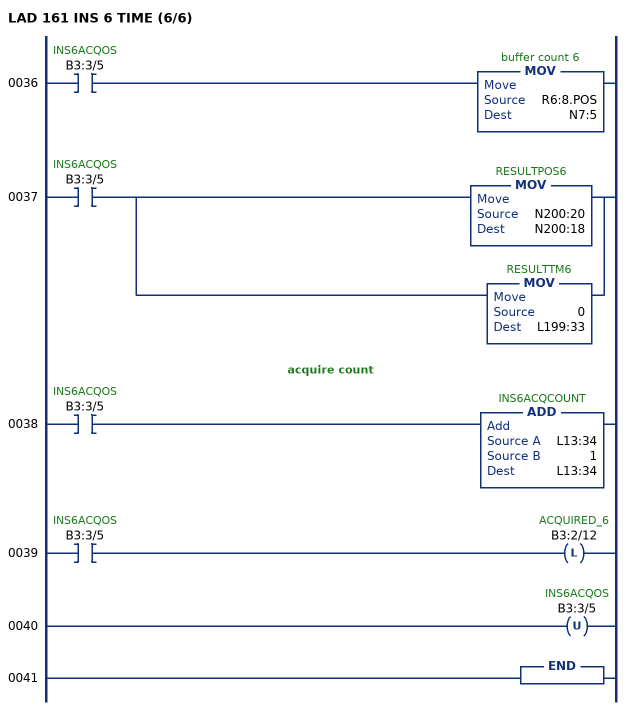
% Rung: 36 %
SOR XIC B3:3/5 MOV R6:8.POS N7:5 EOR
%   B3:3/5  INS6ACQOS %
%   R6:8  "track part location until acquire 6" %
%   N7:5  "buffer count 6" %
% Rung: 37 %
SOR XIC B3:3/5 BST MOV N200:20 N200:18 NXB MOV 0 L199:33 BND EOR
%   B3:3/5  INS6ACQOS %
%   N200:20  ACQPOS6  "part acq pos 6" %
%   N200:18  RESULTPOS6 %
%   L199:33  RESULTTM6 %
% Rung: 38 %
% TITLE: acquire count %
SOR XIC B3:3/5 ADD L13:34 1 L13:34 EOR
%   B3:3/5  INS6ACQOS %
%   L13:34  INS6ACQCOUNT %
% Rung: 39 %
SOR XIC B3:3/5 OTL B3:2/12 EOR
%   B3:3/5  INS6ACQOS %
%   B3:2/12  ACQUIRED_6 %
% Rung: 40 %
SOR OTU B3:3/5 EOR
%   B3:3/5  INS6ACQOS %
% Rung: 41 %
SOR END EOR

LADDER 162 "INS 6 NEW"
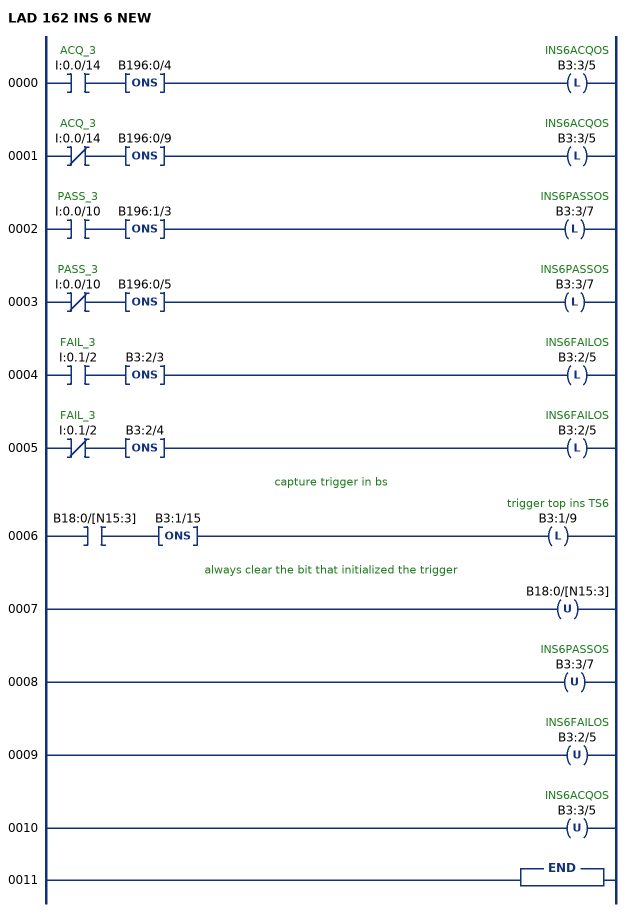
% Rung: 0 %
SOR XIC I:0.0/14 ONS B196:0/4 OTL B3:3/5 EOR
%   I:0.0/14  ACQ_3 %
%   B3:3/5  INS6ACQOS %
% Rung: 1 %
SOR XIO I:0.0/14 ONS B196:0/9 OTL B3:3/5 EOR
%   I:0.0/14  ACQ_3 %
%   B3:3/5  INS6ACQOS %
% Rung: 2 %
SOR XIC I:0.0/10 ONS B196:1/3 OTL B3:3/7 EOR
%   I:0.0/10  PASS_3 %
%   B3:3/7  INS6PASSOS %
% Rung: 3 %
SOR XIO I:0.0/10 ONS B196:0/5 OTL B3:3/7 EOR
%   I:0.0/10  PASS_3 %
%   B3:3/7  INS6PASSOS %
% Rung: 4 %
SOR XIC I:0.1/2 ONS B3:2/3 OTL B3:2/5 EOR
%   I:0.1/2  FAIL_3 %
%   B3:2/5  INS6FAILOS %
% Rung: 5 %
SOR XIO I:0.1/2 ONS B3:2/4 OTL B3:2/5 EOR
%   I:0.1/2  FAIL_3 %
%   B3:2/5  INS6FAILOS %
% Rung: 6 %
% capture trigger in bs %
SOR XIC B18:0/[N15:3] ONS B3:1/15 OTL B3:1/9 EOR
%   N15:3  INS_6_TRIG_LOC %
%   B3:1/9  TS6  "trigger top ins" %
% Rung: 7 %
% always clear the bit that initialized the trigger %
SOR OTU B18:0/[N15:3] EOR
%   N15:3  INS_6_TRIG_LOC %
% Rung: 8 %
SOR OTU B3:3/7 EOR
%   B3:3/7  INS6PASSOS %
% Rung: 9 %
SOR OTU B3:2/5 EOR
%   B3:2/5  INS6FAILOS %
% Rung: 10 %
SOR OTU B3:3/5 EOR
%   B3:3/5  INS6ACQOS %
% Rung: 11 %
SOR END EOR

LADDER 170 "PASS BLOW"
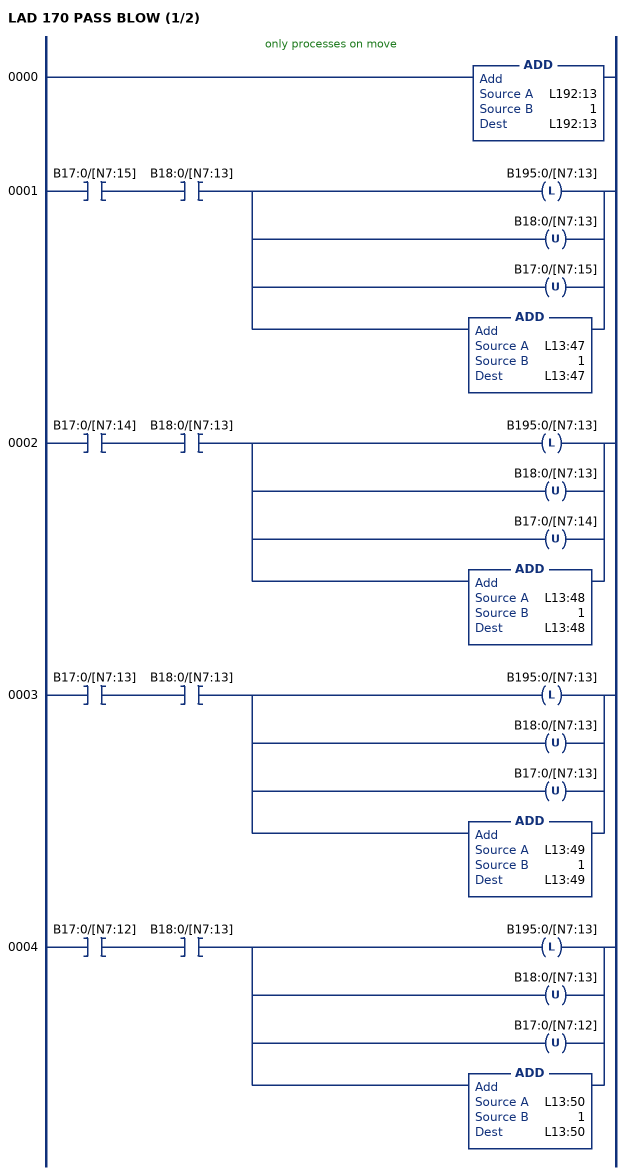
% Rung: 0 %
% only processes on move %
SOR ADD L192:13 1 L192:13 EOR
% Rung: 1 %
SOR XIC B17:0/[N7:15] XIC B18:0/[N7:13] BST OTL B195:0/[N7:13] NXB OTU B18:0/[N7:13] NXB OTU B17:0/[N7:15] NXB ADD L13:47 1 L13:47 BND EOR
%   N7:15  OS5 %
%   N7:13  OS3 %
% Rung: 2 %
SOR XIC B17:0/[N7:14] XIC B18:0/[N7:13] BST OTL B195:0/[N7:13] NXB OTU B18:0/[N7:13] NXB OTU B17:0/[N7:14] NXB ADD L13:48 1 L13:48 BND EOR
%   N7:14  OS4 %
%   N7:13  OS3 %
% Rung: 3 %
SOR XIC B17:0/[N7:13] XIC B18:0/[N7:13] BST OTL B195:0/[N7:13] NXB OTU B18:0/[N7:13] NXB OTU B17:0/[N7:13] NXB ADD L13:49 1 L13:49 BND EOR
%   N7:13  OS3 %
% Rung: 4 %
SOR XIC B17:0/[N7:12] XIC B18:0/[N7:13] BST OTL B195:0/[N7:13] NXB OTU B18:0/[N7:13] NXB OTU B17:0/[N7:12] NXB ADD L13:50 1 L13:50 BND EOR
%   N7:12  OS2 %
%   N7:13  OS3 %

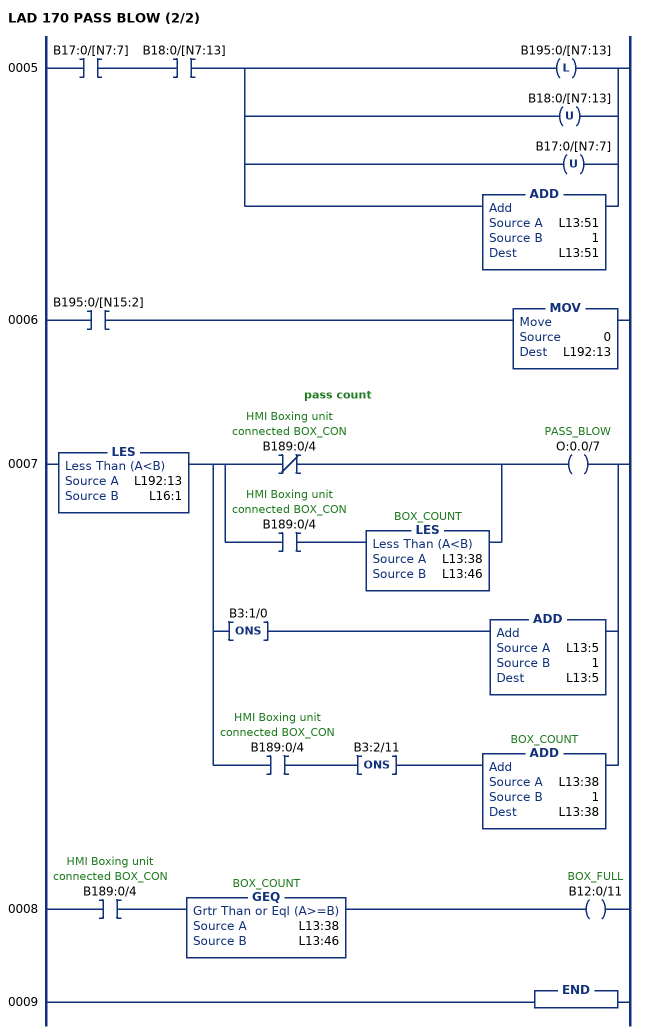
% Rung: 5 %
SOR XIC B17:0/[N7:7] XIC B18:0/[N7:13] BST OTL B195:0/[N7:13] NXB OTU B18:0/[N7:13] NXB OTU B17:0/[N7:7] NXB ADD L13:51 1 L13:51 BND EOR
%   N7:7  OS1 %
%   N7:13  OS3 %
% Rung: 6 %
SOR XIC B195:0/[N15:2] MOV 0 L192:13 EOR
%   N15:2  BLOW_PT %
% Rung: 7 %
% TITLE: pass count %
SOR LES L192:13 L16:1 BST BST XIO B189:0/4 NXB XIC B189:0/4 LES L13:38 L13:46 BND OTE O:0.0/7 NXB ONS B3:1/0 ADD L13:5 1 L13:5 NXB XIC B189:0/4 ONS B3:2/11 ADD L13:38 1 L13:38 BND EOR
%   L16:1  BLOW_TIME %
%   B189:0/4  BOX_CON  "HMI Boxing unit connected" %
%   L13:38  BOX_COUNT %
%   L13:46  BOX_LIMIT  "box count setpoint" %
%   O:0.0/7  PASS_BLOW %
% Rung: 8 %
SOR XIC B189:0/4 GEQ L13:38 L13:46 OTE B12:0/11 EOR
%   B189:0/4  BOX_CON  "HMI Boxing unit connected" %
%   L13:38  BOX_COUNT %
%   L13:46  BOX_LIMIT  "box count setpoint" %
%   B12:0/11  BOX_FULL %
% Rung: 9 %
SOR END EOR

LADDER 180 "RATE"
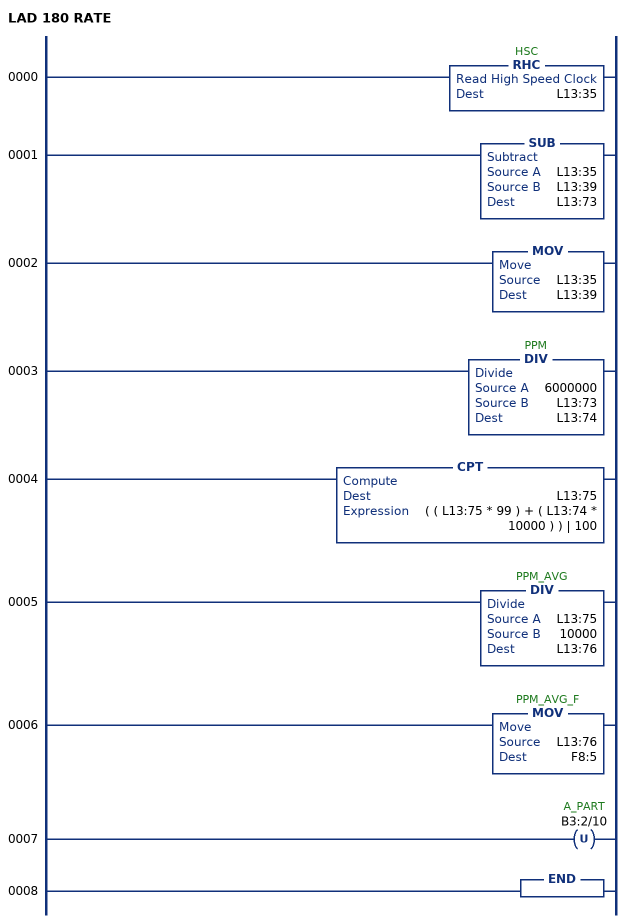
% Rung: 0 %
SOR RHC L13:35 EOR
%   L13:35  HSC %
% Rung: 1 %
SOR SUB L13:35 L13:39 L13:73 EOR
%   L13:35  HSC %
% Rung: 2 %
SOR MOV L13:35 L13:39 EOR
%   L13:35  HSC %
% Rung: 3 %
SOR DIV 6000000 L13:73 L13:74 EOR
%   L13:74  PPM %
% Rung: 4 %
SOR CPT L13:75 " ( ( L13:75 * 99 ) + ( L13:74 * 10000 ) ) | 100 " EOR
%   L13:74  PPM %
% Rung: 5 %
SOR DIV L13:75 10000 L13:76 EOR
%   L13:76  PPM_AVG %
% Rung: 6 %
SOR MOV L13:76 F8:5 EOR
%   L13:76  PPM_AVG %
%   F8:5  PPM_AVG_F %
% Rung: 7 %
SOR OTU B3:2/10 EOR
%   B3:2/10  A_PART %
% Rung: 8 %
SOR END EOR

OTHER DOCUMENTED ADDRESSES
  B3:4/12  "trig 1 event"
  B3:5/1  "placeholder"
  B3:8/1  "bypass extra trigger camera 2"
  B3:8/2  "bypass extra trigger camera 3"
  B3:8/3  "bypass extra trigger camera 4"
  B3:8/6  "a bypass bit"
  B3:8/7  "a bypass bit"
  B3:8/12  "start bottom top camera responce"
  B3:8/13  "extra blow signal for testing"
  B3:8/15  "start side camera responce"
  B3:9/2  "one shot"
  B3:9/4  "start top camera responce"
  B3:9/6  "C1D"
  B3:9/7  "C1t"
  B3:9/8  "C2D"
  B3:9/9  "C2t"
  B3:9/14  "input from hmi to reset count"
  B3:10/0  "bypass part too close"
  B3:10/2  "One Shot"
  B3:10/3  "One Shot"
  B3:10/4  "changing Box chute door operation"
  B3:10/5  "one shot"
  B3:10/6  "excessive data output time"
  B3:10/9  "one shot"
  B3:10/10  "one shot"
  B3:10/11  "bottom part present trailling edge"
  B3:10/13  "one shot"
  B3:10/14  "Dont use"
  B3:10/15  "Reserved For Shift Registers"
  B3:11/0  "bypass unused portion of code"
  B3:11/1  "bypass"
  B3:11/2  "Enable encoder belt movement simulation when testing"
  B3:11/3  "Block blow signals while changing box"
  B3:11/4  "one shot"
  B3:11/6  "one shot"
  B3:11/7  "one shot"
  B3:11/8  "one shot"
  B3:11/11  "one shot"
  B3:11/12  "one shot"
  B3:11/15  "one shot"
  B3:12/0  "one shot"
  B3:12/1  "one shot"
  B3:12/2  "Command 2 Oneshot"
  B3:12/3  "Command 2 Active"
  B3:12/4  "Command3 Oneshot"
  B3:12/5  "Command 3 Active"
  B3:12/6  "Inspection Command Counter"
  B3:12/7  "Command 4 Active"
  B3:12/8  "Command 4 Oneshot"
  B3:12/14  "flip flop bit"
  B3:13/5  "bypass"
  B3:13/6  "Off"
  B3:13/7  "On"
  B3:13/8  "On"
  B3:13/9  "Off"
  B3:13/10  "On"
  B3:13/11  "Off"
  B3:13/12  "Test Trigger to laser Spacing"
  B3:13/15  "Test Signals"
  B3:17/12  "Always Off"
  B9:0/0  "Trigger Insert Position"
  B9:0/1  "bottom of top conveyor part transfer location"
  B9:0/[N7:0]  "Side Camera Trigger Posistion"
  B9:0/[N7:2]  "Mask Start Position"
  B9:0/[N7:6]  "Blow Off Position"
  B9:0/[N7:20]  "part present bit shift load position"
  B9:0/[N7:48]  "Top Camera Trigger Posistion"
  B9:0/[N16:0]  "Trigger Position"
  B9:0/[N17:8]  "part from bottom belt present at top belt optic position"
  B10:0/0  "Pass Insert Position"
  B10:0/[N7:2]  "Pass Bit Position"
  B10:0/[N7:4]  "Pass Insert Position"
  B10:0/[N7:5]  "Pass Start Position"
  B10:0/[N7:6]  "Pass Position"
  B10:0/[N16:4]  "Pass Insert Position"
  B10:0/[N16:6]  "Pass Position"
  B11:0/0  "Trigger Insert Position"
  B11:0/[N7:8]  "Fail Bit Position"
  B11:0/[N16:0]  "Trigger Position"
  B12:1/0  "Conveyor Start Oneshot"
  B12:1/1  "Feed Start Oneshot"
  B12:1/2  "Conveyor Stop Oneshot"
  B12:1/3  "Feed Stop Oneshot"
  B12:1/5  "Conveyor Start Oneshot"
  B12:10  BULK_PACK
  B14:0/0  "Bottom Pass Insert"
  B14:0/4  "Bottom Pass Insert Position"
  B14:0/[N13:14]  "Start Laser Pass"
  B14:0/[N16:4]  "Pass Insert Position"
  B14:0/[N16:6]  "Pass Position"
  B15:0  "Alarm Bits"
  B18:1/1  "bottom pass one shot transfer"
  B18:3/2  "Part Present Oneshot"
  B18:3/3  "Part Present Oneshot"
  B18:5/11  "Transfer bottom pass result from end of bottom conveyor"
  B18:10/15  "Reserved For Shift Registers"
  B18:142  "fack camerea pass signal"
  B22:0  "Transfer Shift Register"
  B22:0/0  "load top conveyor bitshift from bottom cammera pass."
  B22:0/[N17:8]  "bottom good part at top optic position"
  B23:0/[N7:0]  "Bottom Pass Output"
  B185:0/0  "bypass"
  B185:0/1  "bypass"
  B185:0/9  "result time 1 okay"
  B185:0/11  "test fail out"
  B185:0/12  "enable"
  B185:0/13  "enable"
  B185:1/0  "enable"
  B185:1/3  "enable"
  B185:1/7  "enable"
  B191:1/0  "Part measured wider then the limit set in the optic test"
  B191:1/1  "part to part spacing smaller then the set minimum value"
  B191:1/2  "Boxing conveyor backed up"
  B191:2/0  "bottom to top alignment"
  B196:0/13  "waiting for result"
  B196:0/14  "acquire before result os"
  B196:0/15  "enable count"
  B196:1/5  "switch me to EN_1"
  B196:1/9  "Enable alignment Signal"
  B196:1/11  "enable"
  B196:1/12  "enable"
  B196:1/15  "transfer trigger for position alignment logical one shot"
  B196:2/0  "enable"
  B196:2/2  "enable"
  B196:2/8  "enable count"
  B196:2/9  "time out 1"
  B196:2/10  "Reset bad head fault"
  B196:4/0  "test trigger signal 1"
  B196:4/4  "real part within distance of virtual part"
  B196:4/15  "pass in bit shift"
  F8:0  "part to part time us as a float"
  F8:13  "error top"
  F8:15  "error bottom"
  F8:20  "bot belt speed average in pulses per second"
  F8:26  "Part bits loaded into BitShift"
  F8:28  "momentary rate in ppm"
  F8:29  "Count of signals passed to the blow valve"
  F8:31  "Count of off alignment between top and bottom ALIGN_FAILS"
  F8:34  "count of blow signals"
  F8:35  "rate difference"
  F8:38  "averaged rate"
  F8:40  "absoloute difference top"
  F8:41  "absoloute difference bottom"
  F8:42  "Total fail and missed count CAM_NON_PASS"
  F8:43  "change in part rate as %"
  F8:44  "difference as a ratio of the total"
  F8:45  "TOO_CLOSE_BOT"
  F8:46  "TOO_WIDE_BOT"
  F8:48  "transfer"
  F8:49  "TOO_CLOSE_TOP"
  F8:51  "TOO_WIDE_TOP"
  F8:52  "OPTO_FAILS"
  F8:53  "optic fail count top camera TOP_OPT_FAIL_CT"
  F8:54  "optic fail count bot camera BOT_OPT_FAIL_CT"
  F19:4  "Conveyor Input Blip Counter"
  F188:1  "HMI Recerk speed input"
  F188:2  "HMI input for feed wheel speed"
  F188:3  "HMI input for feeder speed"
  F188:4  "HMI input for hopper speed"
  F192:0  "temp"
  F205:0  "feed wheel"
  F205:1  "feed bowl"
  F205:2  "hopper"
  HSC:0.0  "top"
  HSC:0.3/6  "Underflow interrupt"
  HSC:0.3/7  "Overflow interrupt"
  HSC:1.0  "bot"
  HSC:1.3/6  "Underflow interrupt"
  HSC:1.3/7  "Overflow interrupt"
  I:0.0/0  "Encoder Signal "A""
  I:0.0/1  "Encoder Signal "B""
  I:0.0/4  "Encoder Signal "A""
  I:0.0/5  "Encoder Signal "B""
  I:0.0/11  PASS_4
  I:0.0/15  ACQ_4
  I:0.1/3  FAIL_4
  I:0.2/3  "Packaging Conveyor full"
  I:0.2/4  "Packaging Conveyor Box in Position"
  I:0.4  "Spare Analog Input 1"
  I:0.5  "Spare Analog Input 2"
  I:0.6  "Spare Analog Input 3"
  I:2.0/1  REAR_ESTOP
  I:2.0/8  "front door signal"
  I:2.0/9  "rear door signal"
  I:2.0/10  "Maintenance Key Switch"
  I:2.0/12  "input from customer Packager Concluded"
  L13:37  "last part to part time"
  L13:40  "last part time"
  L13:42  "last part to current time"
  L23:1  MPCE_ON
  L23:19  TOP_OPT_FAIL_CT
  L23:34  AIR_PRESSURE_FAULT
  L183:2  "simulated part width"
  L187:5  "pass transfer out signals"
  L187:6  "NoErr transfer out signals"
  L187:7  "ins 1 trigger count"
  L190:0  "count of bottom optic width fails"
  L190:1  "count of gap fails"
  L190:2  "I1 blocked triggers"
  L190:4  "count of parts rejected because acquire time ran out"
  L190:5  "count of parts that received a pass signal but previously failed 1"
  L190:6  "count of result signals received with no part present 1"
  L190:7  "count of results received after maximim time reached"
  L190:8  "pass count"
  L190:9  "fail count"
  L190:10  "acquisition count"
  L190:11  "acquisition without result count"
  L190:12  "count of parts results that time out"
  L190:27  "optic alignment pass signal"
  L190:28  "optic alignment fail signal"
  L190:31  "something wrong, can't happen"
  L190:32  "Crazy wrong, can't happen"
  L192:1  BOT_LAST_TIME  "rtc bot belt previous movement event time"
  L192:2  BOT_CYCLE_TIME  "rtc bot belt time between events"
  L192:16  TOP_LAST_TIME  "rtc top belt previous movement event time"
  L192:17  TOP_CYCLE_TIME  "rtc top belt time between events"
  L201:5  "ms since trig 1 is initialized"
  L201:10  "movement from virtual (pos, add)"
  L204:13  "This optic signal time"
  L204:14  "Last optic signal time"
  L204:15  "time between optic signals"
  N10:1  "old ConveyorStatus"
  N10:2  "PowerOn"
  N10:3  "Local Mode On BypassBoxingPLC"
  N10:4  "Boxing Connected Signal"
  N10:5  "BoxJamSignal"
  N10:6  "WaittingOnBoxSig"
  N10:7  "ConveyorFullSig"
  N10:8  "MachineFaultSig"
  N10:9  "Counter Sensor Fault"
  N10:11  "Feeder Track Sensor Blocked"
  N10:12  "Air Pressure Fault"
  N13:0  "Part Inspecting"
  N13:4  "Completed Counter"
  N13:5  "Trigger Position Counter"
  N13:6  "BlowOff Start Counter"
  N13:7  "BlowOff Stop Counter"
  N13:8  "Inspection Command Counter"
  N13:9  "Complete Counter"
  N13:10  "Pass Signal Counter"
  N13:11  "Solenoid Signal Counter"
  N13:12  "Hold Pass Counter"
  N13:13  "Hold Pass Length"
  N16:1  "Bottom Inspection Offset For Tracking"
  N16:3  "Bit Shift Preset"
  N17:5  "Parts In Tube Counter"
  N17:6  "Parts In Tube Limit"
  N17:9  "Bot to Top Transfer Position"
  N17:12  "Trigger to laser Counter"
  N197:1  "maximim acquire time 1"
  N197:5  "Feeder Speed Output Setting"
  N197:10  "pulse distance to keep blow on then turn off feed"
  N197:11  "speed in pps"
  N197:12  "seconds of ontime"
  N197:20/0  "Deformed Head Blowoff Bit to TOP PLC"
  O:0.0/1  "spare"
  O:0.0/5  INS_4_TRIG
  O:0.0/6  "spare"
  O:0.0/11  "Spare"
  O:0.5  "spare"
  O:3.0/0  "Ready-Run signal to Boxer? Always on unless fault?"
  O:3.0/2  "Customers pecies counting done signal (Change Box?)"
  O:3.0/6  RED_LT  "Red Light"
  O:3.0/7  "Spare"
  O:3.0/8  "spare"
  PFILE:6  "check for part jams"
  PFILE:10  "Bottom belt HSC"
  PFILE:12  "Top belt HSC"
  Q2:55  END_OF_MAIN
  Q5:94  END_OF_BELTS
  R6:5.POS  "Empty Fifo"
  R21:0  "Trigger Shift Register"
  T20:0  "Trigger On Time"
  U:5  "conveyor"
  U:9  "slow data"
  U:11  "transfered data calcuations from the high speed section"
  U:28  "faults"
  U:29  "speed"
  U:30  "count"
  U:31  "rate calc"
  U:32  "boxer"
  U:33  "bulk pack"
  U:34  "customer boxing unit signals"
  U:35  "cleanup"
  U:95  "HMI interface"
  U:120  "simulate part injection"
  U:121  "bot optic"
  U:140  "top optic"

COMMENTS NOT ATTACHED TO A CURRENT RUNG
  F8:13: *************************
    Loads Side Camera Passing data into a bit shift
    *************************
    
    loads passing data bit into passing data bit shift register at the part present cl.
  I:0.0/8: special rung for testing. This rung can simulate a pass signal. It will not be timed correctly.
  B23:0/0: Yet another bit shift load with data in the part position indicating that there was a bottom system part pass as well as a top system part present at this location.
    
    verified works w/bypassed 071910 and unbypassed 072010
  N7:25: 1050
  C5:4: tempory counting to verify pass part count with boxing part count.
  B22:0/0: ***********************
     Bottom Part Syncronizing Logic
    ***********************
    
    This is the point at the bottom of the top conveyor where the part jumps from the bottom conveyor.  This system will then track the part through the top system to the point of the laser optic in order to verify that the part in question has passed the bottom inspection.  I believe that we NEED to include FAILING inspections to eliminate the possibility of a out of position part from passing. LW 072010
  T20:2.ACC: This rung is starting a timer that should be activated directly before the laser optic part presense sensor on the top conveyer and should cause the top optic to be ignored if the bottom camera system didn't pass. however other arrangements must be made if the bottom camera isn't going to be used as is the case with a nut inspection.
  T20:2: The timer used to verify that the part that triggered the top laser optic has passed the bottom camer. needs to be count
  N17:8: ****************************************************************************************************************
    I can not find anywhere in the program where the "Test Spacing From Pickup to Trigger is activated indicating to me that this entire function must not be doing anything in this program at this time.
    ****************************************************************************************************************
  B11:0/0: load part present bit shit with one shot data from the part present sensor
  B3:7/9: ************************************
     The next 3 rungs appear to do nothing
    ***********************************
  B3:6/0: make a bit come on indicating that a part that passed the bottom camera is within  range when crossing the top camera.
  B3:6/1: ***********************
    Part Width and  Location
    ***********************
    
    Calculates the position of parts on the top belt by measureing the part width by calculating the number of belt movement pulses that occure when the optic is blocked and then devides that in half and add that to the optic location in the part presnet bit shift when the top optic is cleared.
  N7:45: not fully functional because of part overlap but measurems the camera responce time when part inspections are not overlaping
  B9:0/[N7:47]: Remove any part present signals outside of expected location
  B9:0/[N7:50]: Remove any part present signals outside of expected location
  F19:0: Counter inside of a high speed counter interrupt counts the number of Bit Shifts that need to be processed in order to move the logic with the parts on the conveyor.
  B3:4/14: *****
    Convertion of the optic signal to something stable
    *****
  F8:14: **************
    Bottom Top Camera Trigger
    *************
    
    Trigger Bottom Top Camera
  N10:4: test if boxing is connected
  B3:6/8: ********************************************************************************************************************************
    Box count reached
    Redo all of boxing;
    1. handle box done, change, box not moving, no new box
    2. everything else is situational, i.e. box removed, box not present
    add bulk pack rutine that just stops bowl and doesn't change box.
    ********************************************************************************************************************************
  T4:27: Time to clear shoot
  B3:6/9: Detect fault condition no box present on conveyor
  B3:11/3: After initial delay allow blow two start functioning
  T4:28: Time to close shoot door
  RUNG000150-000011: trigger count
  RUNG000150-000012: wipe stored part data if acq time expires
  RUNG000150-000013: clear data for aquire time expired
  RUNG000150-000014: clear data for time
  RUNG000150-000016: wiped count
  RUNG000150-000018: pass, fail and acquire inputs
  RUNG000150-000025: pass code / Set pass bit in Bit Shift
    captures result position and processing time
    Unlatch pass bit
  RUNG000150-000032: pass count
  RUNG000150-000035: fail count
  RUNG000150-000038: acquire code
  RUNG000150-000039: Grab trigger/acquire position
    Grab acquire time
  RUNG000150-000041: transfer tracked part positon from trigger/acquire to the acquire/result
    capture acquire time
    reset process time
  L14:8: on when ok for run
  L14:3: off when ok to run
  L14:2: off when ok to run
  L14:5: on when ok to run, rear off turns both off
  N7:76: removed relieance on trigger signal
  N197:20/0: Passes deformed head blowoff command to TOP PLC where solenoid output is located.
  N7:47: ***********************************************************************************************************************************************************
    From side
    ***********************************************************************************************************************************************************
    
    removed relieance on trigger signal
  N7:50: ***********************************************************************************************************************************************************
    From top
    ***********************************************************************************************************************************************************
    
    removed relieance on trigger signal
  B3:10/1: prevents momentary signals from box present sensor from tripping the logic for box not present
    
    This is in responce to a problem created by the sensor occasionally turning on as if no box was in its path when there is a box present.
  B3:6/2: IF PROCESSING FAULT OCURES AT COUNTER SENSOR; CLEAR THE BELT OF PASSING DATA
  L14:23: ****************  nEEDS fIXING  **********************
  L14:36: ****************  nEEDS fIXING  **********************
  RUNG000010-000014: ****
                      Zeros out the non passing part count when one passes
    ****
  RUNG000010-000018: Remove any part present signals outside of expected location
  RUNG000125-000014: clear data for time
  RUNG000125-000013: clear data for aquire time expired
  RUNG000125-000012: wipe stored part data if acq time expires
  RUNG000125-000011: trigger count
  RUNG000125-000007: Trigger output
  RUNG000125-000029: Set pass bit in Bit Shift
    captures result position and processing time
    Unlatch pass bit
  RUNG000125-000027: transfer tracked part positon from trigger/acquire to the acquire/result
    capture acquire time
    reset process time
  RUNG000125-000026: Grab trigger/acquire position
    Grab acquire time
  RUNG000125-000025: pass code / Set pass bit in Bit Shift
    captures result position and processing time
    Unlatch pass bit
  RUNG000125-000018: pass, fail and acquire inputs
  RUNG000125-000016: wiped count
  N7:46: Remove any part present signals outside of expected location

REVISION NOTES
  13: updated count reset
  14: added io moduals
  15: multiple steps toward new hmi integration
  21: test

DATA TABLE (non-zero values as saved)
DATA B3
% B3:0 % 0X8021 0X0030 0X5048 0X9100 0X8304 0X2000 0X02C1 0X0020 0X4007 0X0000
% B3:10 % 0X2041 0X0846 0X2000 0X0000
DATA T4
% .PRE .ACC %
% T4:0 % 300 300
% T4:1 % 150 0
% T4:2 % 32765 0
% T4:3 % 32765 0
% T4:4 % 32765 0
% T4:5 % 150 150
% T4:6 % 5555 32766
% T4:7 % 300 0
% T4:8 % 300 0
% T4:9 % 50 49
% T4:10 % 200 200
% T4:12 % 50 0
% T4:13 % 222 0
% T4:14 % 222 0
% T4:15 % 180 0
% T4:16 % 222 0
% T4:17 % 300 0
% T4:18 % 8 0
% T4:19 % 6 0
% T4:20 % 10 0
% T4:21 % 100 0
% T4:22 % 20 0
% T4:23 % 900 0
% T4:24 % 1000 0
% T4:25 % 250 250
% T4:26 % 666 666
% T4:27 % 400 0
% T4:28 % 400 0
% T4:29 % 10 0
% T4:30 % 50 50
% T4:31 % 20 0
% T4:32 % 69 0
DATA R6
% .LEN .POS %
% R6:0 % 3 0
% R6:1 % 3 0
% R6:2 % 3 0
% R6:3 % 3 0
% R6:4 % 1250 0
% R6:5 % 1250 0
% R6:6 % 1650 0
% R6:7 % 435 0
% R6:8 % 3 0
% R6:9 % 3 0
% R6:10 % 659 0
% R6:11 % 659 0
% R6:12 % 10 0
% R6:13 % 10 0
% R6:14 % 10 0
% R6:15 % 10 0
% R6:16 % 1650 0
% R6:17 % 659 0
% R6:18 % 659 0
DATA N7
% N7:0 % 6 1224 3 996 0 2 1 1611 92 75
% N7:10 % 1216 61 1610 1609 1608 1607 3 3 1222 1242
% N7:20 % 3 3 183 0 0 0 -403 0 0 0
% N7:50 % 1236 0 175 16 0 0 0 1464 12 0
% N7:60 % 1 32767 4012 20 31 0 0 15 30 20
% N7:70 % 0 21 23 27738 32767 0 122 0 16 0
% N7:80 % 0 6 95 0 0 0 5 500 0 0
% N7:90 % 2011 4 4 12 1 0 0 0 0 1600
% N7:100 % 123 124 1227 1228 1237 1238 0 0 0 0
% N7:110 % 0 0 0 0 0 0 0 0 400 0
% N7:120 % 25007 61 0 0 0 0 0 0 0 0
DATA F8
% F8:0 % 12536 206.64 23807 499 0.23807
% F8:5 % 257 0 500 1.9 210
% F8:10 % 0.0888 0.08897486 2364 101 63.26563
% F8:15 % 37.73437 4040 210 0 0
% F8:20 % 0 0.02 0 1 0
% F8:25 % 0 932781 0.222 279.6551 848597
% F8:30 % 0 170 0.03 38 852060
% F8:35 % 0 0 0 0 77
% F8:40 % 101 37.73437 0 100 1
% F8:45 % 1 2 0.21455 0 0
% F8:50 % 0 0 1 0 1
% F8:55 % 2000000 -221 0 0 0
% F8:95 % 0 0 0 492 4.92
DATA B9
% B9:130 % 0X0000 0X0000 0X0000 0X0000 0X2000 0X0000 0X0000 0X0000 0X0000 0X8000
% B9:140 % 0X2480 0X0000 0X0000 0X0000 0X0000 0X0000 0X0000 0X0000 0X0000 0X0000
% B9:160 % 0X0000 0X0000 0X0000 0X0000 0X0000 0X0000 0X2000 0X0002 0X0000 0X0000
% B9:170 % 0X0000 0X0000 0X0000 0X2000 0X0000 0X0000 0X0000 0X0000 0X0000 0X0000
% B9:180 % 0X0000 0X0000 0X0000 0X0000 0X0000 0X0002 0X0000 0X0000 0X0000 0X0000
% B9:190 % 0X0010 0X0000 0X0000 0X0000 0X0000 0X0000 0X0000 0X0000 0X0000 0X0000
% B9:200 % 0X2B64 0X2B64 0X0000 0X0010 0X0000 0X2000 0X0000 0X0000 0X0000 0X0000
% B9:220 % 0X0000 0X0000 0X0000 0X0200 0X0000 0X0000 0X0000 0X0000 0X0000 0X0020
% B9:230 % 0X0040 0X0000 0X0000 0X0000 0X0000 0X0000 0X0000 0X0000 0X0000 0X0000
DATA B11
% B11:180 % 0X0000 0X8000 0X0000 0X0000 0X0000 0X0000 0X0000 0X0000 0X0000 0X0000
% B11:240 % 0X0000 0X0000 0X0000 0X4000 0X0000 0X0000 0X0000 0X0000 0X0000 0X0000
DATA B12
% B12:0 % 0X0155 0X0000 0X0000 0X0000 0X0000 0X0000 0X0000 0X0000 0X0000 0X0000
DATA L13
% L13:0 % 308402300 308407124 4824 0 1000
% L13:5 % 86255 7 2 1162124017 1162124017
% L13:10 % 492 90891 87436 92135 92044
% L13:15 % 282802241 -2147483648 2147483647 2147483647 82058
% L13:20 % 18816300 18813411 5 5 281643860
% L13:25 % 18757058 65520 100 4693 1142
% L13:30 % 154 153 92034 303 92131
% L13:35 % -436115285 489 12536 0 -436115285
% L13:40 % -867278648 677 12536 900728 32089
% L13:45 % 816709 100 10 6 4854661
% L13:50 % 5 5 250 100000 250
% L13:55 % 13 22 0 0 15
% L13:60 % 100000 100 0 0 0
% L13:65 % 0 0 317148919 317148142 281709380
% L13:70 % 317175733 317175698 35 1768218 3
% L13:75 % 2565908 257 0 0 0
DATA F14
% F14:0 % 50.08958 47.95059 5 5 1212.342
% F14:5 % 7863.84 13106.4 982.98 0 0
DATA N15
% N15:0 % 6 908 1612 1224 1212 170 103 1204 1004 5555
% N15:10 % 62 620 0 0 0 0 1204 0 0 0
DATA L16
% L16:0 % 8 9 5 5 5
% L16:5 % 250 5000 5000 182 19
% L16:10 % 1256 18 2045 40 98
% L16:15 % 99 0 0 0 0
DATA B17
% B17:100 % 0X0000 0X0000 0X0000 0X0000 0X0000 0X0000 0X0800 0X0000 0X1000 0X0000
% B17:110 % 0X4000 0X0000 0X0000 0X0000 0X0000 0X0000 0X0000 0X0000 0X0000 0X0000
% B17:120 % 0X0000 0X0000 0X0000 0X0000 0X0000 0X0000 0X0000 0X2000
DATA B18
% B18:100 % 0X0000 0X0000 0X0000 0X0000 0X0000 0X0001 0X0000 0X0080 0X0000 0X8240
% B18:110 % 0X0000 0X0400 0X0000 0X0000 0X0000 0X0000 0X0040 0X0000 0X0000 0X0010
% B18:120 % 0X0000 0X0000 0X0000 0X0000 0X0000 0X0000 0X0000 0X2000
DATA L23
% L23:0 % 65535 -65536 -65536 -65536 -65536
% L23:5 % -65536 -65536 212 65535 -65536
% L23:10 % -65536 0 17 10 17
% L23:15 % 0 0 0 0 8
% L23:20 % 0 -65536 -65536 -65536 -65536
% L23:25 % -65536 20 19 20 0
% L23:30 % 0 0 -65536 -65536 -65536
% L23:35 % -65536 -65536 -65536 -65536 -65536
% L23:40 % 16270 18414 0 63266 -65536
% L23:45 % 5062 0 0 0 0
% L23:50 % 0 -65536 -65536 17 -65536
% L23:55 % 33 5079 -65536 0 0
% L23:60 % 0 -65536 -65536 -65536 0
DATA L24
% L24:0 % -65536 122 -65536 222 -65536
% L24:5 % 65535 -65536 -65536 -65536 -65536
% L24:10 % 50 27 0 1 23
% L24:15 % 1198 1030 95 18 30
% L24:20 % 30 -65536 1226 -65536 -65536
% L24:25 % 222 1236 -65536 -65536 222
% L24:30 % 1466 27 10000 -65536 55
% L24:35 % 180 -65536 180 65535 101
% L24:40 % 101 1000 -65536 -65536 10
% L24:45 % 222 192 -65536 0 -65536
% L24:50 % -999 30 10000 65535 900
DATA L42
% L42:0 % -65536 0 0 0 0
% L42:5 % 45 45 45 0 0
% L42:20 % 0 0 32766 32766 0
% L42:50 % 0 30
DATA L183
% L183:0 % 999 216325420 12 1000000000 0
% L183:5 % 101 80 59 0 0
DATA B185
% B185:0 % 0X0200 0X0001 0X0000 0X0000 0X0000 0X0000 0X0000 0X0000 0X0000 0X0000
DATA N186
% N186:0 % 100 0 0 0 0 0 0 0 0 0
DATA L187
% L187:0 % 34 26 35 0 0
% L187:5 % 1063 0 0 0 0
DATA F188
% F188:0 % 6 66 11 44 29
DATA B189
% B189:0 % 0X00E0 0X0000 0X0000 0X0000 0X0000 0X0000 0X0000 0X0000 0X0000 0X0000
DATA L190
% L190:0 % 1 5 0 0 0
% L190:30 % 0 2 0 0 0
DATA B191
% B191:0 % 0X0000 0X0001 0X0000 0X0000 0X0000 0X0000 0X0000 0X0000 0X0000 0X0000
DATA L192
% L192:0 % 317333597 266932201 5055 16 0
% L192:5 % 100000 2500000 999 999 8
% L192:10 % 0 0 0 392500 17
% L192:15 % 317332943 332250347 860888 15 0
% L192:20 % 180 2600000 0 0 0
DATA F193
% F193:0 % 0.9304597 0.315 0.022 6 50
% F193:5 % 0.2081299 0.14 0.02913818 46.52299 1524.372
% F193:10 % 0.011 0.195 0.165 0.337 50
% F193:15 % 0.2801514 0.18 0.05042725 59.55566 1951.401
DATA B196
% B196:0 % 0X0816 0X9FFE 0X0005 0X0000 0X0000 0X0000 0X0000 0X0000 0X0000 0X0000
% B196:30 % 0XE800 0X9BFF 0XEBFF 0XFFDF 0XFFFF 0X0000 0X0000 0X0000 0X0000 0X0000
DATA N197
% N197:0 % 1560 150 1111 2500 2500 14417 5555 300 150 0
% N197:10 % 4000 969 4 0 0 0 0 0 0 0
% N197:30 % 15 48 0 0 0 0 0 0 0 0
DATA B198
% B198:0 % 0X0009 0X0000 0X0000 0X0000 0X0000 0X0000 0X0000 0X0000 0X0000 0X0000
DATA L199
% L199:0 % 1 5571998 134 11 3579521
% L199:5 % 0 0 0 5 221042
% L199:10 % 0 224 10256 280 0
% L199:15 % 0 0 0 278717848 518
% L199:20 % 28295 16430853 5001 5001 0
% L199:25 % 0 0 28329 1 1131572
% L199:30 % 1131837 251 1159715 1159802 111
% L199:35 % 555 555 0 0 0
DATA N200
% N200:0 % 2046 2047 2046 2047 2045 1224 1004 2045 2045 2045
% N200:10 % 0 0 0 1277 178 2046 1000 2045 2045 1218
% N200:20 % 1232 0 0 0 0 0 0 0 0 0
% N200:30 % 0 0 32767 0 0 0 0 0 0 0
DATA L201
% L201:0 % 20 40 40 -3011735 44
% L201:5 % 96629277 0 0 -3010662 0
% L201:10 % 0 0 0 327 43
% L201:15 % 0 43 0 43 36830
DATA B202
% B202:0 % 0X2241 0X0000 0X0001 0X0000 0X0000 0X0000 0X0000 0X0000 0X0000 0X0000
DATA N203
% N203:0 % 115 115 116 333 334 333 444 0 445 444
% N203:10 % 555 556 555 0 0 0 0 0 0 0
DATA L204
% L204:0 % 111 101 111 1362 124
% L204:5 % 2000 2000 1784 222 0
% L204:10 % 0 0 0 1327077052 1327077052
% L204:15 % 1327077052 1327077052 1 0 0
% L204:20 % 0 0 33 0 0
% L204:30 % 33 0 0 0 0
DATA F205
% F205:0 % 655.32 655.32 655.32 655.32 0
